///Emulation modes for the virtual sensor
{attribute 'qualified_only'}
{attribute 'strict'}
{attribute 'to_string'}
(**************************************************************************************
 *  Application     :   BoxControl Framework
 *  Revision date   :   $Date: 2021-04-09 08:29:02 +0200 (fre, 09 apr 2021) $
 *  Author          :   CDC
 * ------------------------------------------------------------------------------------
 *  © Swisslog AG
 *  Swisslog is not liable for any usage of this source code that is not agreed 
 *  on between Swisslog and the other party. The mandatory legal liability remains 
 *  unaffected.
 * ------------------------------------------------------------------------------------
 *  Revision History: 
 *
 *  VERSION DATE         INITIALS     DESCRIPTION
 *  0.0     DD.MM.YYYY   (name)       (explain customized modifications)
 *
 **************************************************************************************)
TYPE E_SensorEmulateModes :
(
	VIRTUAL,
    PREVIOUS,
    NEXT,
    OWN
);
END_TYPE

(* stored: Version 1.1.0.1, ProductVersion 3.1.4024.4
   EnumerationTextList E_SensorEmulateModes: Id {d9a83c43-949b-4170-8b57-028c5a4b7f6b} *)
